(* Logix 5000 project; controller STAT 1756-L72 rev 20.12; software revision 20.04; part 13 of 34 *)
(* tags used below, declared in another part *)
   P21 : BOOL;
   P22 : BOOL;
   B14 : DINT[30];
   B16 : DINT[30];
   B17 : DINT[30];
   B3 : DINT[256];
   B9 : DINT[40];
   F8 : REAL[256];
   FL_STOP_RO : BOOL;
   I10_000_Bit00 : ALIAS FOR I10[0].0;   // Drukknop start CL7 P 19A
   I10_000_Bit01 : ALIAS FOR I10[0].1;   // Drukknop stop CL7 P 19A
   I10_000_Bit02 : ALIAS FOR I10[0].2;   // Drukknop start CL7 P 19B
   I10_000_Bit03 : ALIAS FOR I10[0].3;   // Drukknop stop CL7 P 19B
   I10_001_Bit07 : ALIAS FOR I10[1].7;   // Hand Automaat CL9
   I10_001_Bit08 : ALIAS FOR I10[1].8;   // Drukknop start P9 CL9
   I10_001_Bit09 : ALIAS FOR I10[1].9;   // Drukknop stop P7 CL9
   I10_001_Bit10 : ALIAS FOR I10[1].10;   // Drukknop start P8 CL9
   I10_001_Bit11 : ALIAS FOR I10[1].11;   // Drukknop stop P8 CL9
   I10_001_Bit12 : ALIAS FOR I10[1].12;   // Drukknop start P9 CL9
   I10_001_Bit13 : ALIAS FOR I10[1].13;   // Drukknop stop P9 CL9
   I19_000_Bit00 : ALIAS FOR I19[0].0;   // VANNE ALIBERT OUVERTE
   I19_000_Bit01 : ALIAS FOR I19[0].1;   // VANNE ALIBERT FERMEE
   I1_005_Bit15 : ALIAS FOR I1[5].15;
   I1_016_Bit06 : ALIAS FOR I1[16].6;   // CL2 start res.
   I2_000_Bit04 : ALIAS FOR I2[0].4;   // Deelnoodstop cl6 eurowater
   I2_000_Bit06 : ALIAS FOR I2[0].6;   // Deelnoodstop cl7 IBT B
   I3_000_Bit09 : ALIAS FOR I3[0].9;   // Motor pro 1 voedingpomp osmose 1 in driehoek
   I3_000_Bit10 : ALIAS FOR I3[0].10;   // Motor pro 1 voedingpomp osmose 1 in ster
   I3_000_Bit13 : ALIAS FOR I3[0].13;   // Motor pro 2 voedingpomp osmose 2 in driehoek
   I3_000_Bit14 : ALIAS FOR I3[0].14;   // Motor pro 2 voedingpomp osmose 2 in ster
   I3_001_Bit01 : ALIAS FOR I3[1].1;   // Motor p21 kuip az in driehoek
   I3_001_Bit02 : ALIAS FOR I3[1].2;   // Motor p21 kuip az in ster
   I3_001_Bit05 : ALIAS FOR I3[1].5;   // Motor p22 kuip az in driehoek
   I3_001_Bit06 : ALIAS FOR I3[1].6;   // Motor p22 kuip az in ster
   I3_001_Bit09 : ALIAS FOR I3[1].9;   // Motor voedingspomp osmose 3 in drie
   I3_001_Bit10 : ALIAS FOR I3[1].10;   // Motor voed osmose 3 ster
   I6_000_Bit10 : ALIAS FOR I6[0].10;   // pressostaat osmose1
   I6_000_Bit11 : ALIAS FOR I6[0].11;   // pressostaat osmose2
   I6_000_Bit12 : ALIAS FOR I6[0].12;   // pressostaat osmose3
   I7_000_Bit08 : ALIAS FOR I7[0].8;   // midden alarm ketel tampon
   I7_000_Bit09 : ALIAS FOR I7[0].9;   // laag alarm ketel tampon
   I8_000_Bit00 : ALIAS FOR I8[0].0;   // niveau kuip az hoog alarm
   I8_000_Bit01 : ALIAS FOR I8[0].1;   // niveau kuip az midden
   I8_000_Bit02 : ALIAS FOR I8[0].2;   // niveau kuip az laag niv
   I8_000_Bit04 : ALIAS FOR I8[0].4;   // niveau kuip 20m hoog alarm
   I8_000_Bit05 : ALIAS FOR I8[0].5;   // niveau midden kuip 20m
   I8_000_Bit06 : ALIAS FOR I8[0].6;   // niveau kuip 20m laag niv
   I8_000_Bit08 : ALIAS FOR I8[0].8;   // laag niveau kuip 1 voorb. polyelectrolute
   I8_000_Bit11 : ALIAS FOR I8[0].11;   // hoog niveau kuip 2 voorb. polyelectrolute
   I8_001_Bit09 : ALIAS FOR I8[1].9;   // Schakelaar hand autom cl6
   I8_001_Bit10 : ALIAS FOR I8[1].10;   // drukknop start cl6 pro1
   I8_001_Bit11 : ALIAS FOR I8[1].11;   // drukknop stop cl6 pro1
   I8_001_Bit12 : ALIAS FOR I8[1].12;   // drukknop start cl6 pro2
   I8_001_Bit13 : ALIAS FOR I8[1].13;   // drukknop stop cl6 pro2
   I8_001_Bit14 : ALIAS FOR I8[1].14;   // drukknop start cl6 p21
   I8_001_Bit15 : ALIAS FOR I8[1].15;   // drukknop stop cl6 p21
   I9_000_Bit00 : ALIAS FOR I9[0].0;   // Drukknop start CL6 P22
   I9_000_Bit01 : ALIAS FOR I9[0].1;   // Drukknop stop CL6 P22
   I9_000_Bit02 : ALIAS FOR I9[0].2;   // Drukknop start CL6 PRO3
   I9_000_Bit03 : ALIAS FOR I9[0].3;   // Drukknop stop CL6 PRO3
   I9_000_Bit04 : ALIAS FOR I9[0].4;   // Drukknop start CL6 P21
   I9_000_Bit05 : ALIAS FOR I9[0].5;   // Drukknop stop CL6 P21
   I9_000_Bit09 : ALIAS FOR I9[0].9;   // Hand_Auto CL7
   I9_001_Bit06 : ALIAS FOR I9[1].6;   // Drukknop start CL7 AG1
   I9_001_Bit07 : ALIAS FOR I9[1].7;   // Drukknop stop CL7 AG1
   I9_001_Bit08 : ALIAS FOR I9[1].8;   // Drukknop start CL7 AG2
   I9_001_Bit09 : ALIAS FOR I9[1].9;   // Drukknop stop CL7 AG2
   I9_001_Bit10 : ALIAS FOR I9[1].10;   // Drukknop start CL7 AG3
   I9_001_Bit11 : ALIAS FOR I9[1].11;   // Drukknop stop CL7 AG3
   N11 : DINT[150];
   N12 : DINT[230];
   N13 : DINT[230];
   O12_000_Bit03 : ALIAS FOR O12[0].3;   // motor ag1 mixer krimp neutralisatie AG1_MIXER_KRIMP
   O12_000_Bit08 : ALIAS FOR O12[0].8;   // pomp ag2 mixer vat 1 AG2_MIXER_VAT1
   O12_000_Bit09 : ALIAS FOR O12[0].9;   // pomp ag3 mixer vat 2 AG3_MIXER_VAT2
   O12_000_Bit12 : ALIAS FOR O12[0].12;   // Motor P19a zuiveringspomp controleweger P19_ZUIVERP
   O12_000_Bit13 : ALIAS FOR O12[0].13;   // Motor P20 zuiveringspomp controleweger P20_ZUIVERP
   O12_001_Bit03 : ALIAS FOR O12[1].3;   // Motor P7 voedingspomp omgekeerde osmose 1 P7_OSMOSE_1
   O12_001_Bit04 : ALIAS FOR O12[1].4;   // Motor P8 voedingspomp omgekeerde osmose 2 P8_OSMOSE_2
   O12_001_Bit05 : ALIAS FOR O12[1].5;   // Motor P9 voedingspomp omgekeerde osmose 3 P9_OSMOSE_3
   O15_001_Bit07 : ALIAS FOR O15[1].7;   // EV3 EV3
   O16_000_Bit00 : ALIAS FOR O16[0].0;   // COMMANDE VANNE ALIBERT
   O18_001_Bit00 : ALIAS FOR O18[1].0;   // pompe 1 puisard ligne 4
   O18_001_Bit01 : ALIAS FOR O18[1].1;   // pompe 2 puisard ligne 4
   O18_001_Bit06 : ALIAS FOR O18[1].6;
   O18_001_Bit07 : ALIAS FOR O18[1].7;   // pomp pompen uit kelder p23
   O18_001_Bit08 : ALIAS FOR O18[1].8;   // pomp pompen uit kelder p24
   P23 : BOOL;
   P24 : BOOL;
   T27 : TIMER[100];
   T4 : TIMER[200];
(* ibt, continued *)

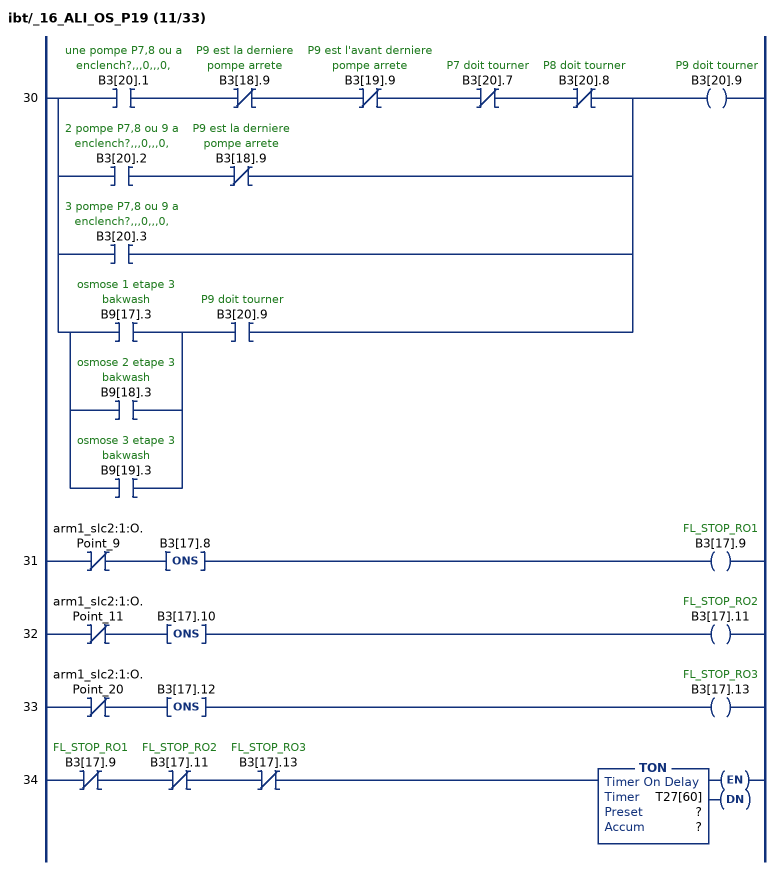
   [picture p202: ibt/_16_ALI_OS_P19 rungs 30-34]
   30: [XIC(B3[20].1) XIO(B3[18].9) XIO(B3[19].9) XIO(B3[20].7) XIO(B3[20].8) ,[XIC(B3[20].2) XIO(B3[18].9) ,XIC(B3[20].3) ] ,[XIC(B9[17].3) ,XIC(B9[18].3) ,XIC(B9[19].3) ] XIC(B3[20].9) ]OTE(B3[20].9);
   31: XIO(arm1_slc2:1:O.Point_9)ONS(B3[17].8)OTE(B3[17].9);
   32: XIO(arm1_slc2:1:O.Point_11)ONS(B3[17].10)OTE(B3[17].11);
   33: XIO(arm1_slc2:1:O.Point_20)ONS(B3[17].12)OTE(B3[17].13);
   34: XIO(B3[17].9)XIO(B3[17].11)XIO(B3[17].13)TON(T27[60],?,?);
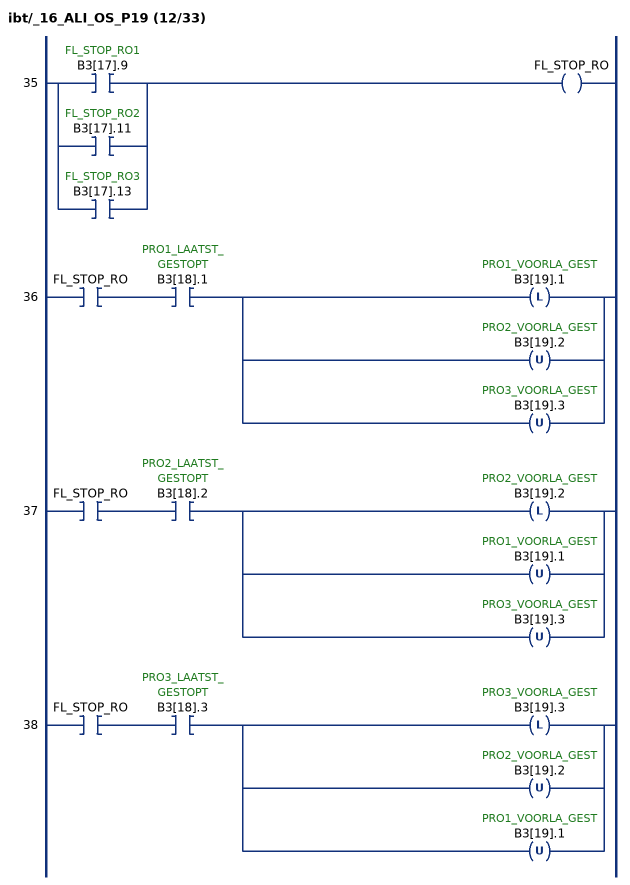
   35: [XIC(B3[17].9) ,[XIC(B3[17].11) ,XIC(B3[17].13) ] ]OTE(FL_STOP_RO);
   36: XIC(FL_STOP_RO)XIC(B3[18].1)[OTL(B3[19].1) ,[OTU(B3[19].2) ,OTU(B3[19].3) ] ];
   37: XIC(FL_STOP_RO)XIC(B3[18].2)[OTL(B3[19].2) ,[OTU(B3[19].1) ,OTU(B3[19].3) ] ];
   38: XIC(FL_STOP_RO)XIC(B3[18].3)[OTL(B3[19].3) ,[OTU(B3[19].2) ,OTU(B3[19].1) ] ];
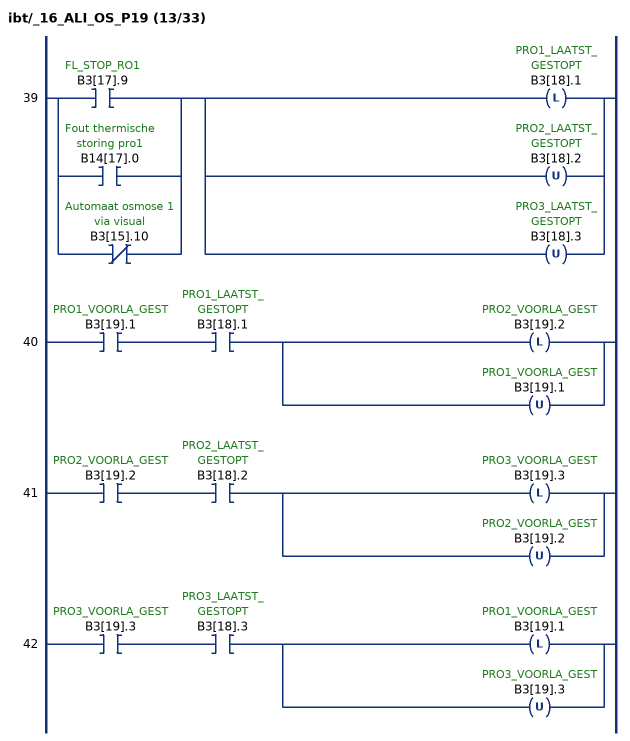
   39: [XIC(B3[17].9) ,[XIC(B14[17].0) ,XIO(B3[15].10) ] ][OTL(B3[18].1) ,[OTU(B3[18].2) ,OTU(B3[18].3) ] ];
   40: XIC(B3[19].1)XIC(B3[18].1)[OTL(B3[19].2) ,OTU(B3[19].1) ];
   41: XIC(B3[19].2)XIC(B3[18].2)[OTL(B3[19].3) ,OTU(B3[19].2) ];
   42: XIC(B3[19].3)XIC(B3[18].3)[OTL(B3[19].1) ,OTU(B3[19].3) ];
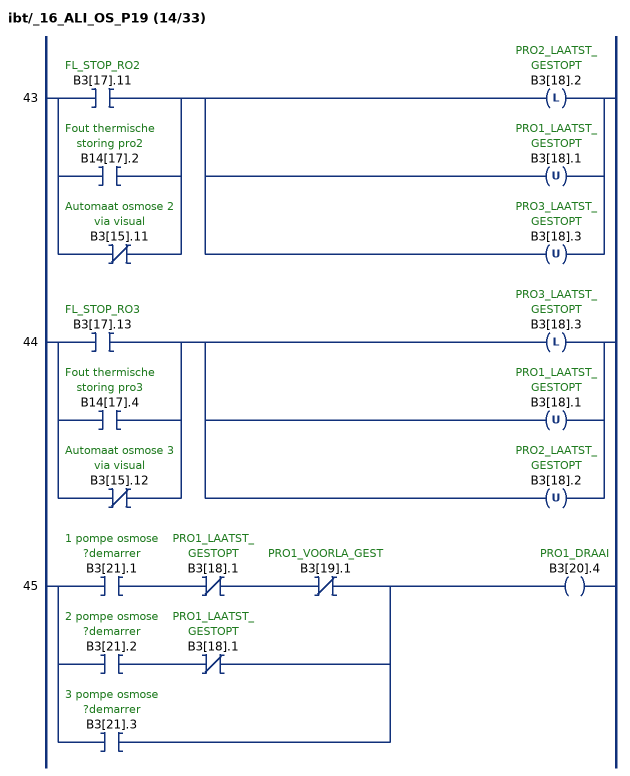
   43: [XIC(B3[17].11) ,[XIC(B14[17].2) ,XIO(B3[15].11) ] ][OTL(B3[18].2) ,[OTU(B3[18].1) ,OTU(B3[18].3) ] ];
   44: [XIC(B3[17].13) ,[XIC(B14[17].4) ,XIO(B3[15].12) ] ][OTL(B3[18].3) ,[OTU(B3[18].1) ,OTU(B3[18].2) ] ];
   45: [XIC(B3[21].1) XIO(B3[18].1) XIO(B3[19].1) ,[XIC(B3[21].2) XIO(B3[18].1) ,XIC(B3[21].3) ] ]OTE(B3[20].4);
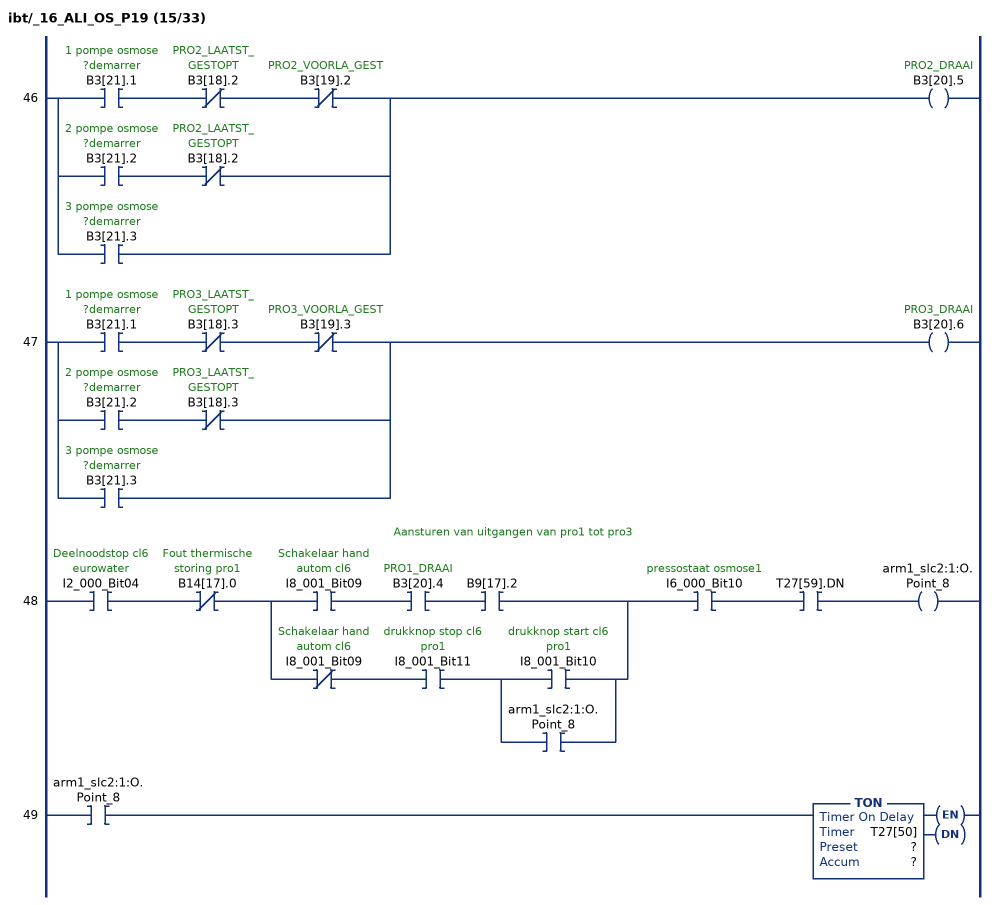
   46: [XIC(B3[21].1) XIO(B3[18].2) XIO(B3[19].2) ,[XIC(B3[21].2) XIO(B3[18].2) ,XIC(B3[21].3) ] ]OTE(B3[20].5);
   47: [XIC(B3[21].1) XIO(B3[18].3) XIO(B3[19].3) ,[XIC(B3[21].2) XIO(B3[18].3) ,XIC(B3[21].3) ] ]OTE(B3[20].6);
   // Aansturen van uitgangen van pro1 tot pro3
   48: XIC(I2_000_Bit04)XIO(B14[17].0)[XIC(I8_001_Bit09) XIC(B3[20].4) XIC(B9[17].2) ,XIO(I8_001_Bit09) XIC(I8_001_Bit11) [XIC(I8_001_Bit10) ,XIC(arm1_slc2:1:O.Point_8) ] ]XIC(I6_000_Bit10)XIC(T27[59].DN)OTE(arm1_slc2:1:O.Point_8);
   49: XIC(arm1_slc2:1:O.Point_8)TON(T27[50],?,?);
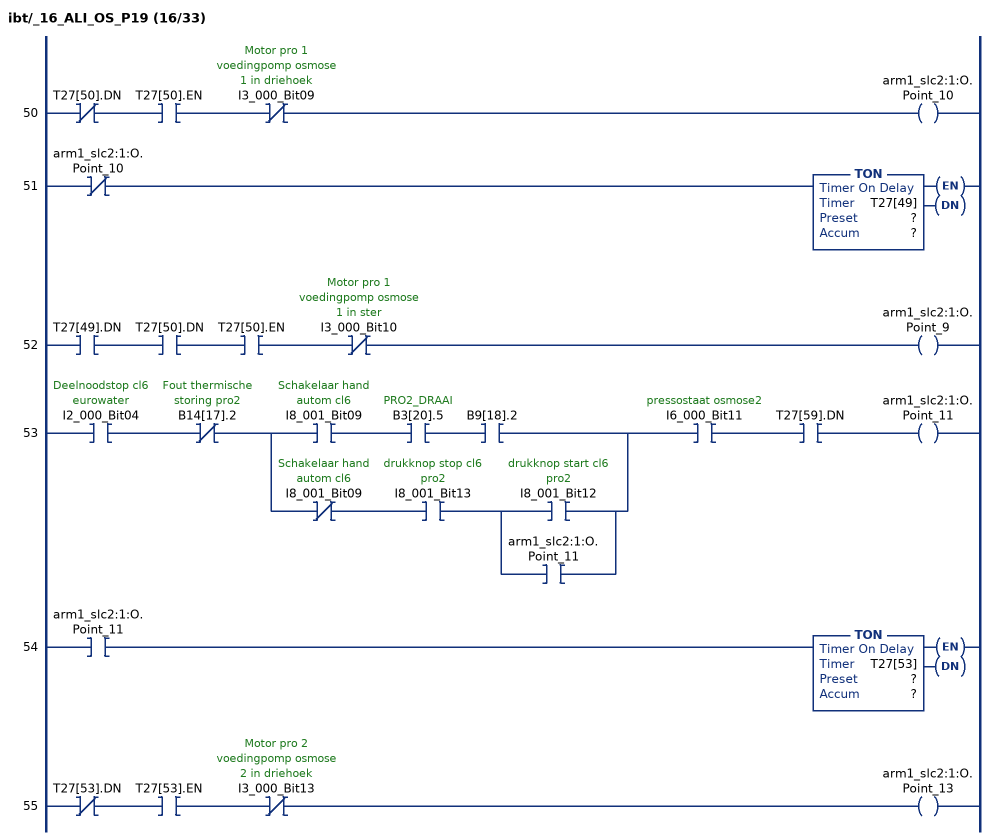
   50: XIO(T27[50].DN)XIC(T27[50].EN)XIO(I3_000_Bit09)OTE(arm1_slc2:1:O.Point_10);
   51: XIO(arm1_slc2:1:O.Point_10)TON(T27[49],?,?);
   52: XIC(T27[49].DN)XIC(T27[50].DN)XIC(T27[50].EN)XIO(I3_000_Bit10)OTE(arm1_slc2:1:O.Point_9);
   53: XIC(I2_000_Bit04)XIO(B14[17].2)[XIC(I8_001_Bit09) XIC(B3[20].5) XIC(B9[18].2) ,XIO(I8_001_Bit09) XIC(I8_001_Bit13) [XIC(I8_001_Bit12) ,XIC(arm1_slc2:1:O.Point_11) ] ]XIC(I6_000_Bit11)XIC(T27[59].DN)OTE(arm1_slc2:1:O.Point_11);
   54: XIC(arm1_slc2:1:O.Point_11)TON(T27[53],?,?);
   55: XIO(T27[53].DN)XIC(T27[53].EN)XIO(I3_000_Bit13)OTE(arm1_slc2:1:O.Point_13);
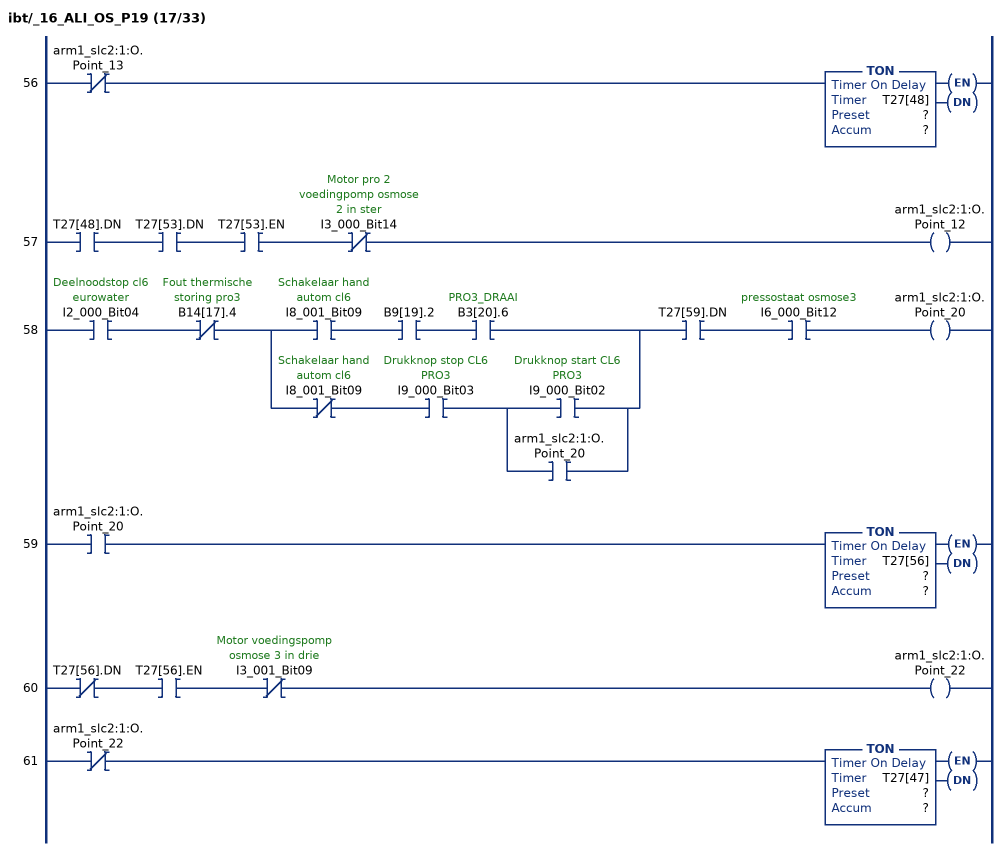
   56: XIO(arm1_slc2:1:O.Point_13)TON(T27[48],?,?);
   57: XIC(T27[48].DN)XIC(T27[53].DN)XIC(T27[53].EN)XIO(I3_000_Bit14)OTE(arm1_slc2:1:O.Point_12);
   58: XIC(I2_000_Bit04)XIO(B14[17].4)[XIC(I8_001_Bit09) XIC(B9[19].2) XIC(B3[20].6) ,XIO(I8_001_Bit09) XIC(I9_000_Bit03) [XIC(I9_000_Bit02) ,XIC(arm1_slc2:1:O.Point_20) ] ]XIC(T27[59].DN)XIC(I6_000_Bit12)OTE(arm1_slc2:1:O.Point_20);
   59: XIC(arm1_slc2:1:O.Point_20)TON(T27[56],?,?);
   60: XIO(T27[56].DN)XIC(T27[56].EN)XIO(I3_001_Bit09)OTE(arm1_slc2:1:O.Point_22);
   61: XIO(arm1_slc2:1:O.Point_22)TON(T27[47],?,?);
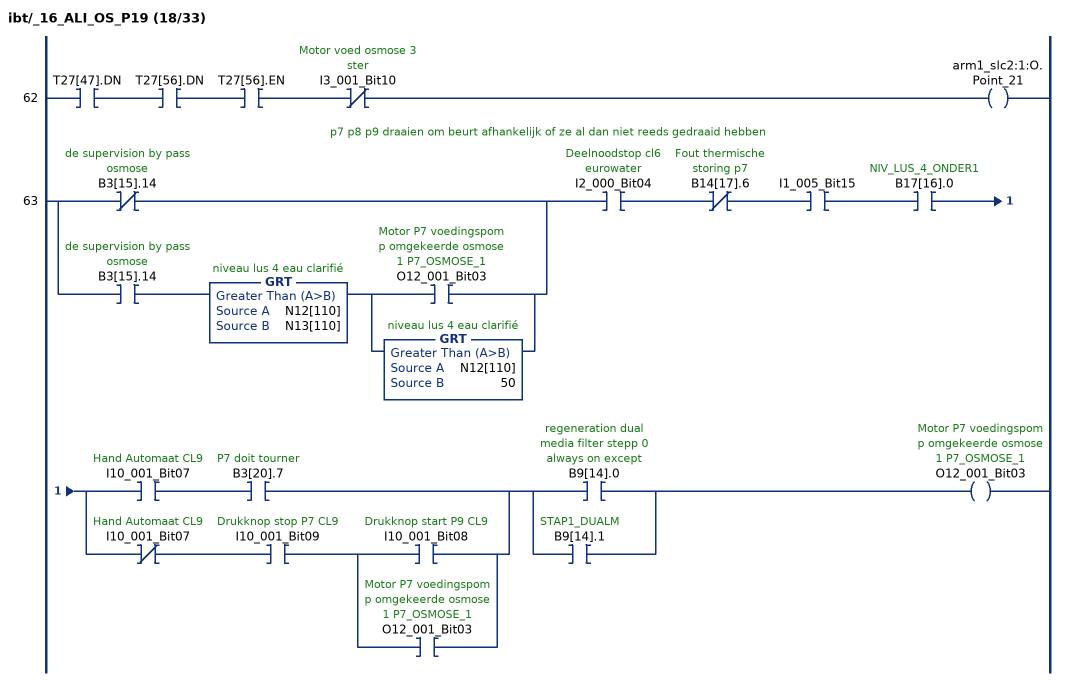
   62: XIC(T27[47].DN)XIC(T27[56].DN)XIC(T27[56].EN)XIO(I3_001_Bit10)OTE(arm1_slc2:1:O.Point_21);
   // p7 p8 p9 draaien om beurt afhankelijk of ze al dan niet reeds gedraaid hebben
   63: [XIO(B3[15].14) ,XIC(B3[15].14) GRT(N12[110],N13[110]) [XIC(O12_001_Bit03) ,GRT(N12[110],50) ] ]XIC(I2_000_Bit04)XIO(B14[17].6)XIC(I1_005_Bit15)XIC(B17[16].0)[XIC(I10_001_Bit07) XIC(B3[20].7) ,XIO(I10_001_Bit07) XIC(I10_001_Bit09) [XIC(I10_001_Bit08) ,XIC(O12_001_Bit03) ] ][XIC(B9[14].0) ,XIC(B9[14].1) ]OTE(O12_001_Bit03);
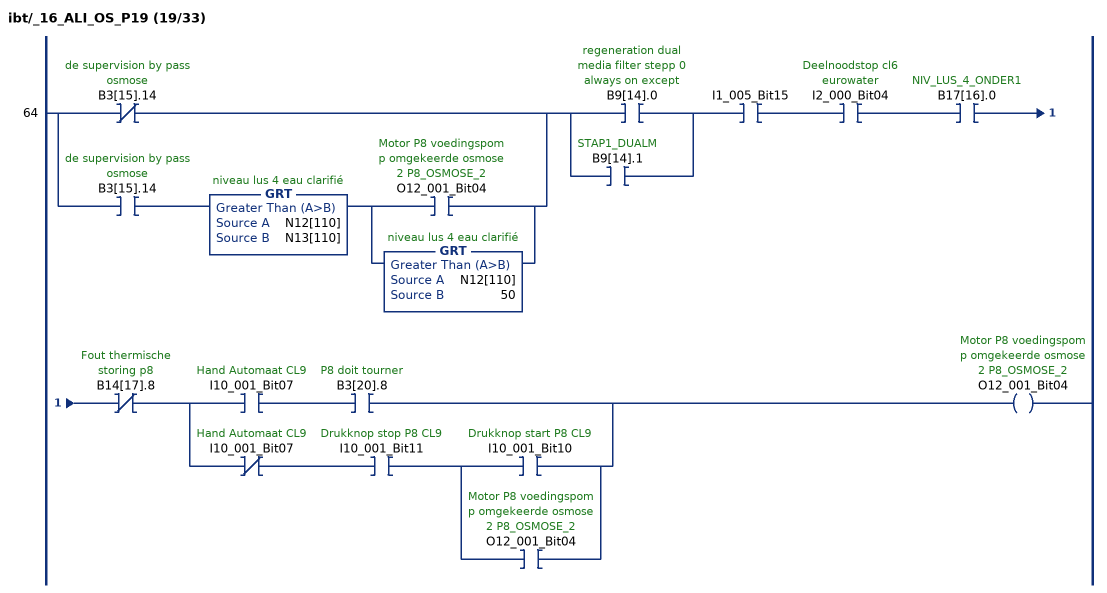
   64: [XIO(B3[15].14) ,XIC(B3[15].14) GRT(N12[110],N13[110]) [XIC(O12_001_Bit04) ,GRT(N12[110],50) ] ][XIC(B9[14].0) ,XIC(B9[14].1) ]XIC(I1_005_Bit15)XIC(I2_000_Bit04)XIC(B17[16].0)XIO(B14[17].8)[XIC(I10_001_Bit07) XIC(B3[20].8) ,XIO(I10_001_Bit07) XIC(I10_001_Bit11) [XIC(I10_001_Bit10) ,XIC(O12_001_Bit04) ] ]OTE(O12_001_Bit04);
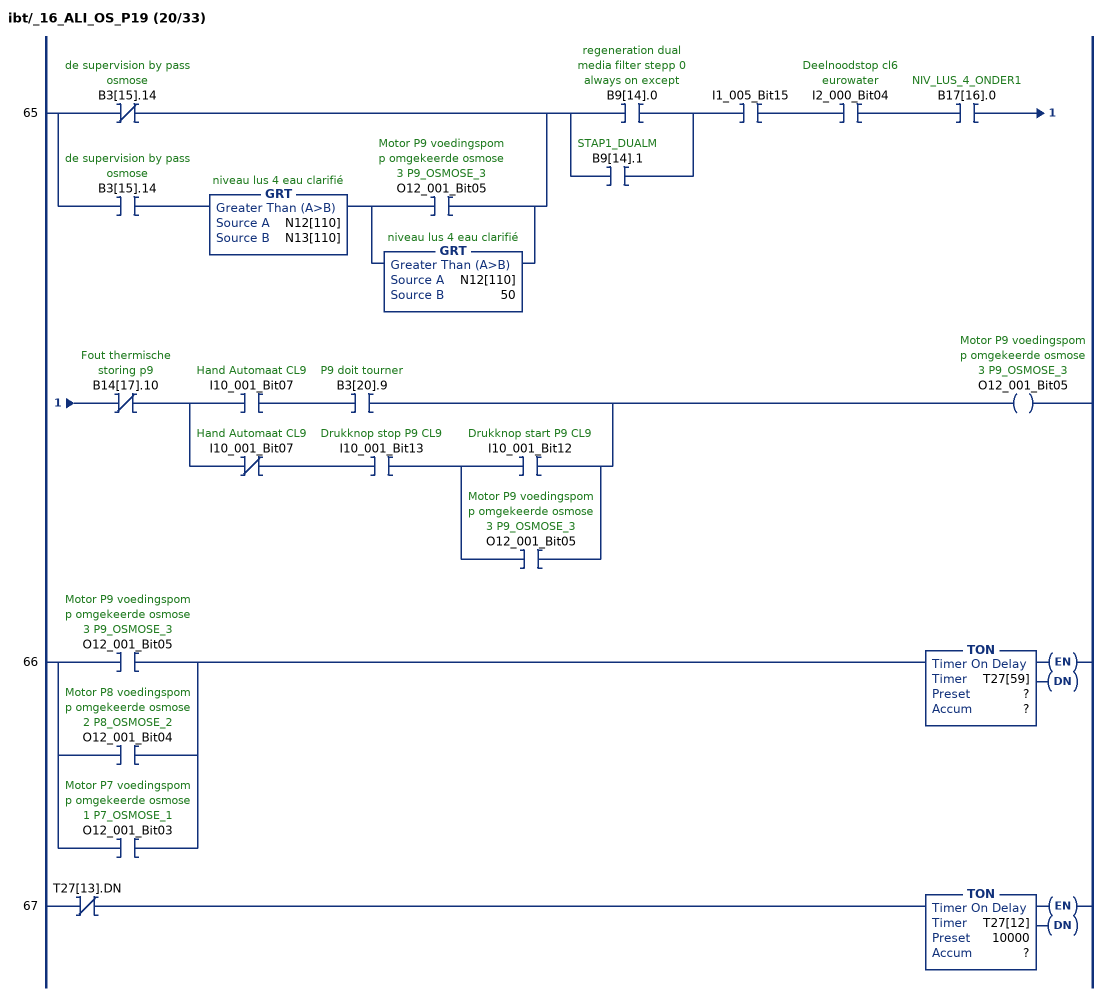
   65: [XIO(B3[15].14) ,XIC(B3[15].14) GRT(N12[110],N13[110]) [XIC(O12_001_Bit05) ,GRT(N12[110],50) ] ][XIC(B9[14].0) ,XIC(B9[14].1) ]XIC(I1_005_Bit15)XIC(I2_000_Bit04)XIC(B17[16].0)XIO(B14[17].10)[XIC(I10_001_Bit07) XIC(B3[20].9) ,XIO(I10_001_Bit07) XIC(I10_001_Bit13) [XIC(I10_001_Bit12) ,XIC(O12_001_Bit05) ] ]OTE(O12_001_Bit05);
   66: [XIC(O12_001_Bit05) ,[XIC(O12_001_Bit04) ,XIC(O12_001_Bit03) ] ]TON(T27[59],?,?);
   67: XIO(T27[13].DN)TON(T27[12],?,?);
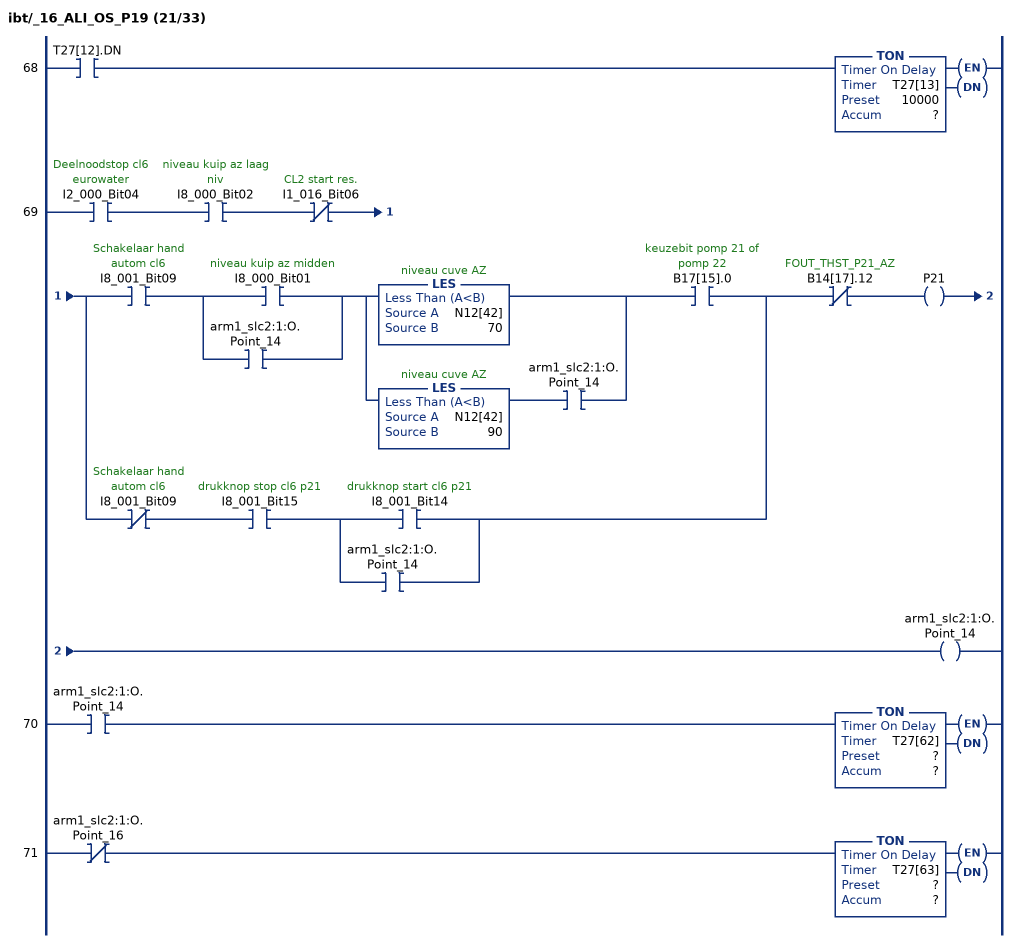
   68: XIC(T27[12].DN)TON(T27[13],?,?);
   69: XIC(I2_000_Bit04)XIC(I8_000_Bit02)XIO(I1_016_Bit06)[XIC(I8_001_Bit09) [XIC(I8_000_Bit01) ,XIC(arm1_slc2:1:O.Point_14) ] [LES(N12[42],70) ,LES(N12[42],90) XIC(arm1_slc2:1:O.Point_14) ] XIC(B17[15].0) ,XIO(I8_001_Bit09) XIC(I8_001_Bit15) [XIC(I8_001_Bit14) ,XIC(arm1_slc2:1:O.Point_14) ] ]XIO(B14[17].12)OTE(P21)OTE(arm1_slc2:1:O.Point_14);
   70: XIC(arm1_slc2:1:O.Point_14)TON(T27[62],?,?);
   71: XIO(arm1_slc2:1:O.Point_16)TON(T27[63],?,?);
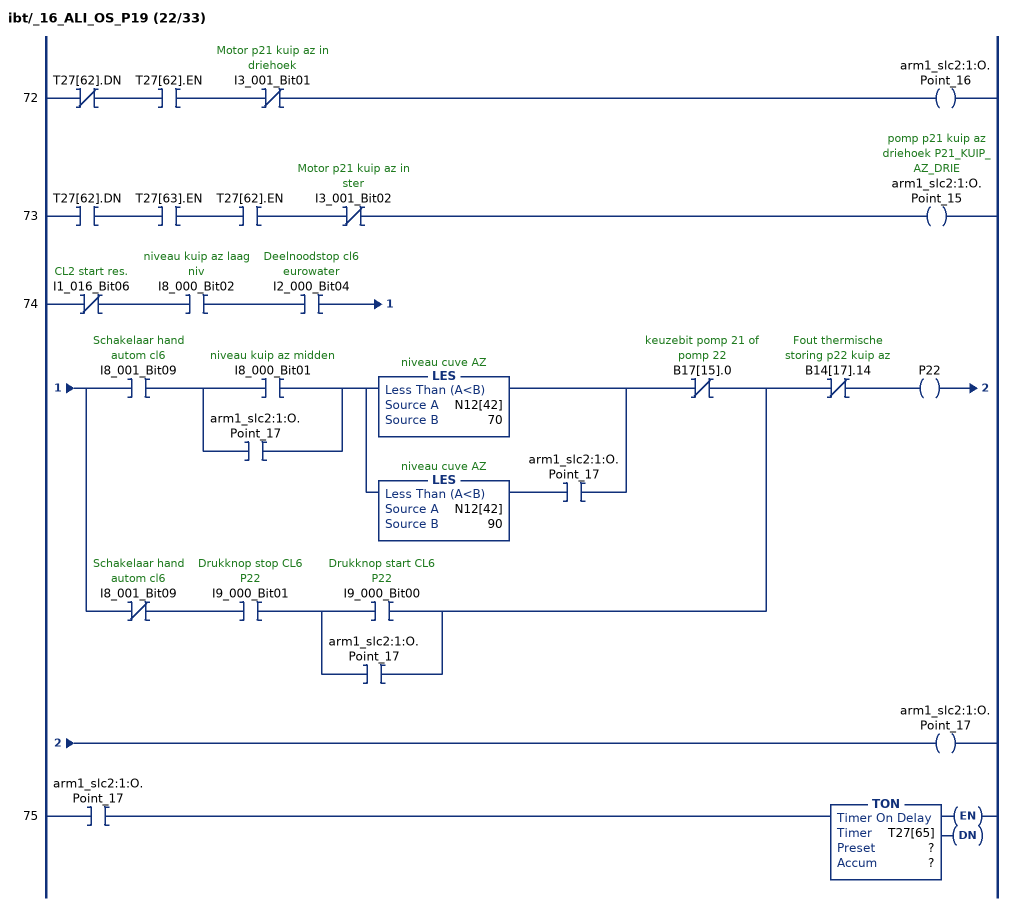
   72: XIO(T27[62].DN)XIC(T27[62].EN)XIO(I3_001_Bit01)OTE(arm1_slc2:1:O.Point_16);
   73: XIC(T27[62].DN)XIC(T27[63].EN)XIC(T27[62].EN)XIO(I3_001_Bit02)OTE(arm1_slc2:1:O.Point_15);
   74: XIO(I1_016_Bit06)XIC(I8_000_Bit02)XIC(I2_000_Bit04)[XIC(I8_001_Bit09) [XIC(I8_000_Bit01) ,XIC(arm1_slc2:1:O.Point_17) ] [LES(N12[42],70) ,LES(N12[42],90) XIC(arm1_slc2:1:O.Point_17) ] XIO(B17[15].0) ,XIO(I8_001_Bit09) XIC(I9_000_Bit01) [XIC(I9_000_Bit00) ,XIC(arm1_slc2:1:O.Point_17) ] ]XIO(B14[17].14)OTE(P22)OTE(arm1_slc2:1:O.Point_17);
   75: XIC(arm1_slc2:1:O.Point_17)TON(T27[65],?,?);
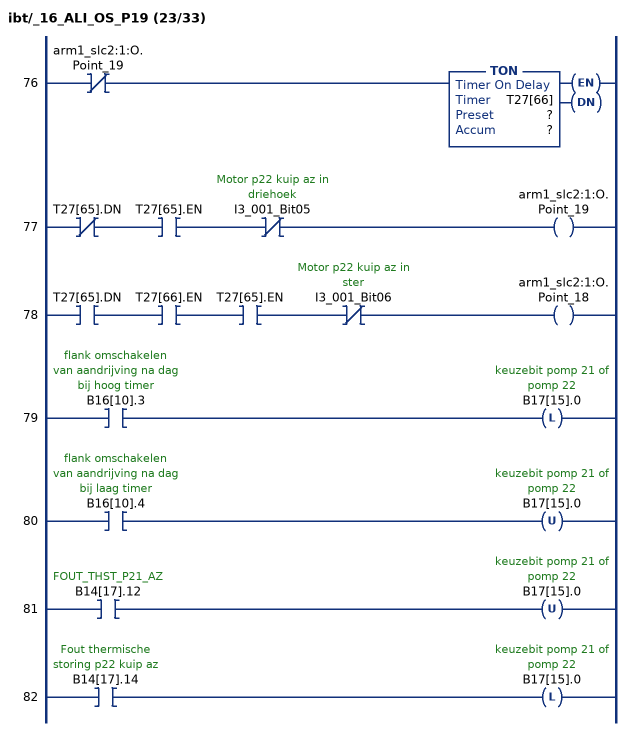
   76: XIO(arm1_slc2:1:O.Point_19)TON(T27[66],?,?);
   77: XIO(T27[65].DN)XIC(T27[65].EN)XIO(I3_001_Bit05)OTE(arm1_slc2:1:O.Point_19);
   78: XIC(T27[65].DN)XIC(T27[66].EN)XIC(T27[65].EN)XIO(I3_001_Bit06)OTE(arm1_slc2:1:O.Point_18);
   79: XIC(B16[10].3)OTL(B17[15].0);
   80: XIC(B16[10].4)OTU(B17[15].0);
   81: XIC(B14[17].12)OTU(B17[15].0);
   82: XIC(B14[17].14)OTL(B17[15].0);
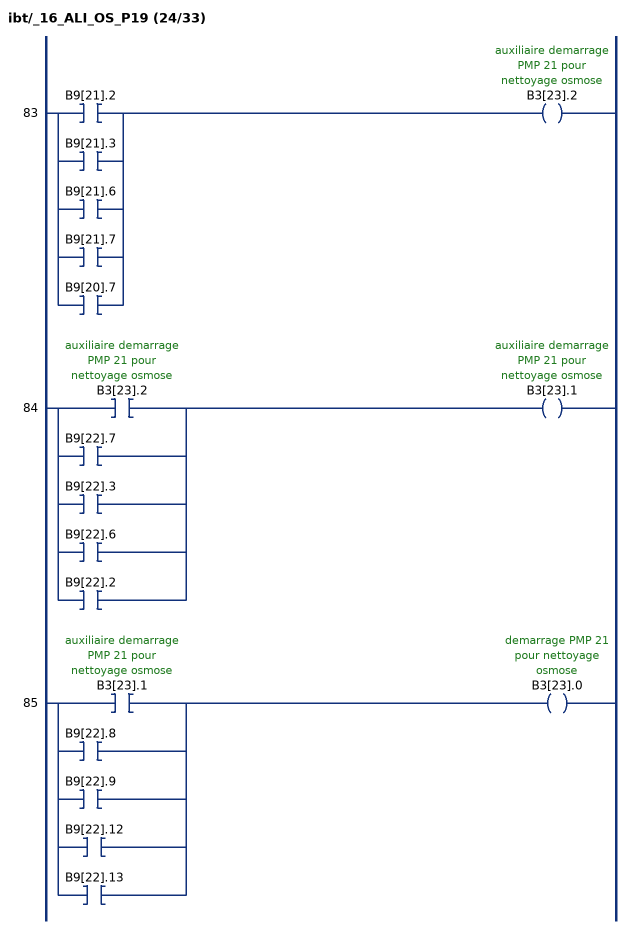
   83: [XIC(B9[21].2) ,XIC(B9[21].3) ,XIC(B9[21].6) ,XIC(B9[21].7) ,XIC(B9[20].7) ]OTE(B3[23].2);
   84: [XIC(B3[23].2) ,XIC(B9[22].7) ,XIC(B9[22].3) ,XIC(B9[22].6) ,XIC(B9[22].2) ]OTE(B3[23].1);
   85: [XIC(B3[23].1) ,XIC(B9[22].8) ,XIC(B9[22].9) ,XIC(B9[22].12) ,XIC(B9[22].13) ]OTE(B3[23].0);
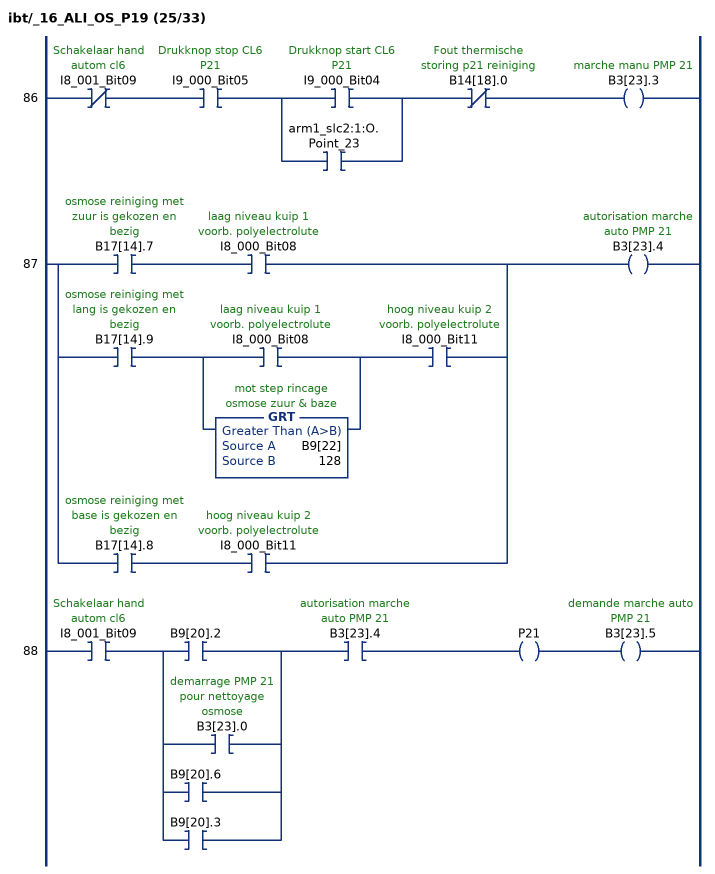
   86: XIO(I8_001_Bit09)XIC(I9_000_Bit05)[XIC(I9_000_Bit04) ,XIC(arm1_slc2:1:O.Point_23) ]XIO(B14[18].0)OTE(B3[23].3);
   87: [XIC(B17[14].7) XIC(I8_000_Bit08) ,XIC(B17[14].9) [XIC(I8_000_Bit08) ,GRT(B9[22],128) ] XIC(I8_000_Bit11) ,XIC(B17[14].8) XIC(I8_000_Bit11) ]OTE(B3[23].4);
   88: XIC(I8_001_Bit09)[XIC(B9[20].2) ,XIC(B3[23].0) ,XIC(B9[20].6) ,XIC(B9[20].3) ]XIC(B3[23].4)OTE(P21)OTE(B3[23].5);
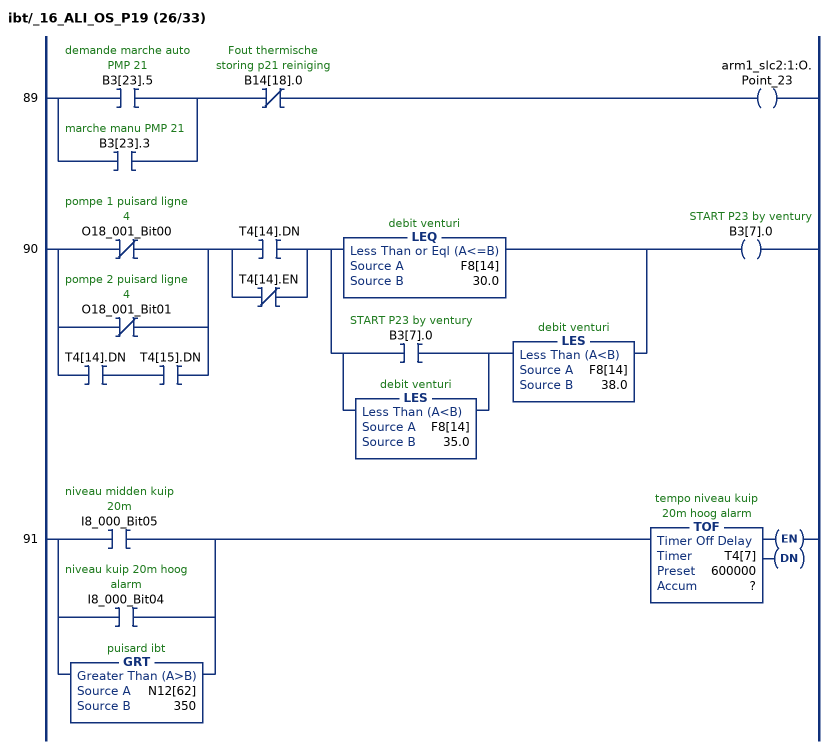
   89: [XIC(B3[23].5) ,XIC(B3[23].3) ]XIO(B14[18].0)OTE(arm1_slc2:1:O.Point_23);
   90: [XIO(O18_001_Bit00) ,XIO(O18_001_Bit01) ,XIC(T4[14].DN) XIC(T4[15].DN) ][XIC(T4[14].DN) ,XIO(T4[14].EN) ][LEQ(F8[14],30.0) ,[XIC(B3[7].0) ,LES(F8[14],35.0) ] LES(F8[14],38.0) ]OTE(B3[7].0);
   91: [XIC(I8_000_Bit05) ,XIC(I8_000_Bit04) ,GRT(N12[62],350) ]TOF(T4[7],?,?);
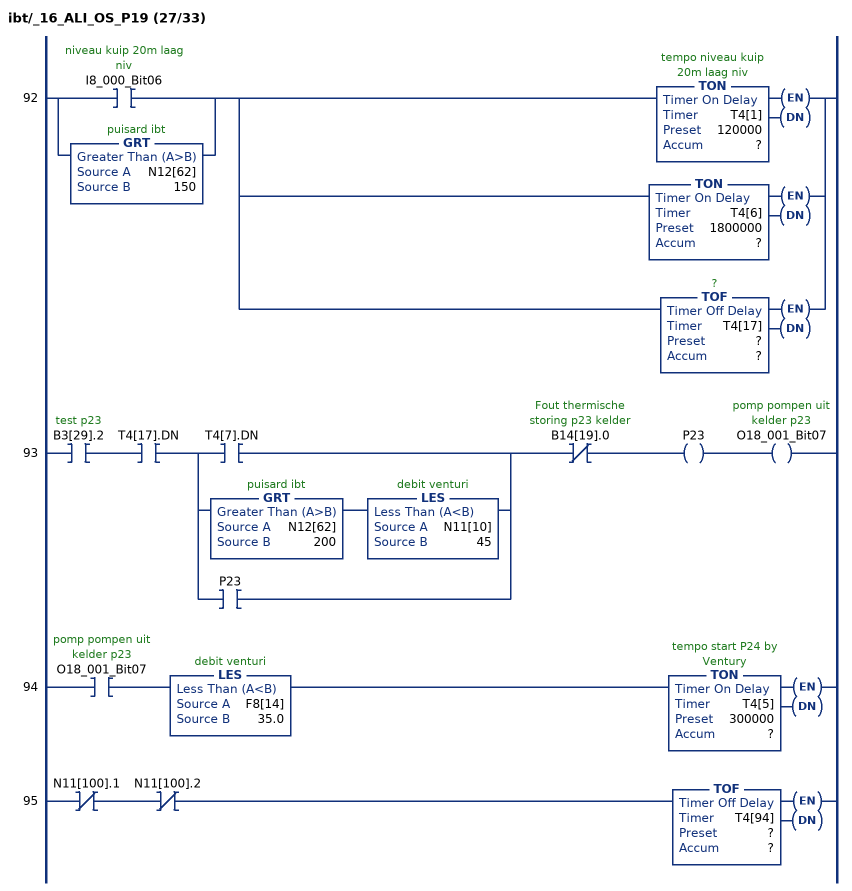
   92: [XIC(I8_000_Bit06) ,GRT(N12[62],150) ][TON(T4[1],?,?) ,TON(T4[6],?,?) ,TOF(T4[17],?,?) ];
   93: XIC(B3[29].2)XIC(T4[17].DN)[XIC(T4[7].DN) ,GRT(N12[62],200) LES(N11[10],45) ,XIC(P23) ]XIO(B14[19].0)OTE(P23)OTE(O18_001_Bit07);
   94: XIC(O18_001_Bit07)LES(F8[14],35.0)TON(T4[5],?,?);
   95: XIO(N11[100].1)XIO(N11[100].2)TOF(T4[94],?,?);
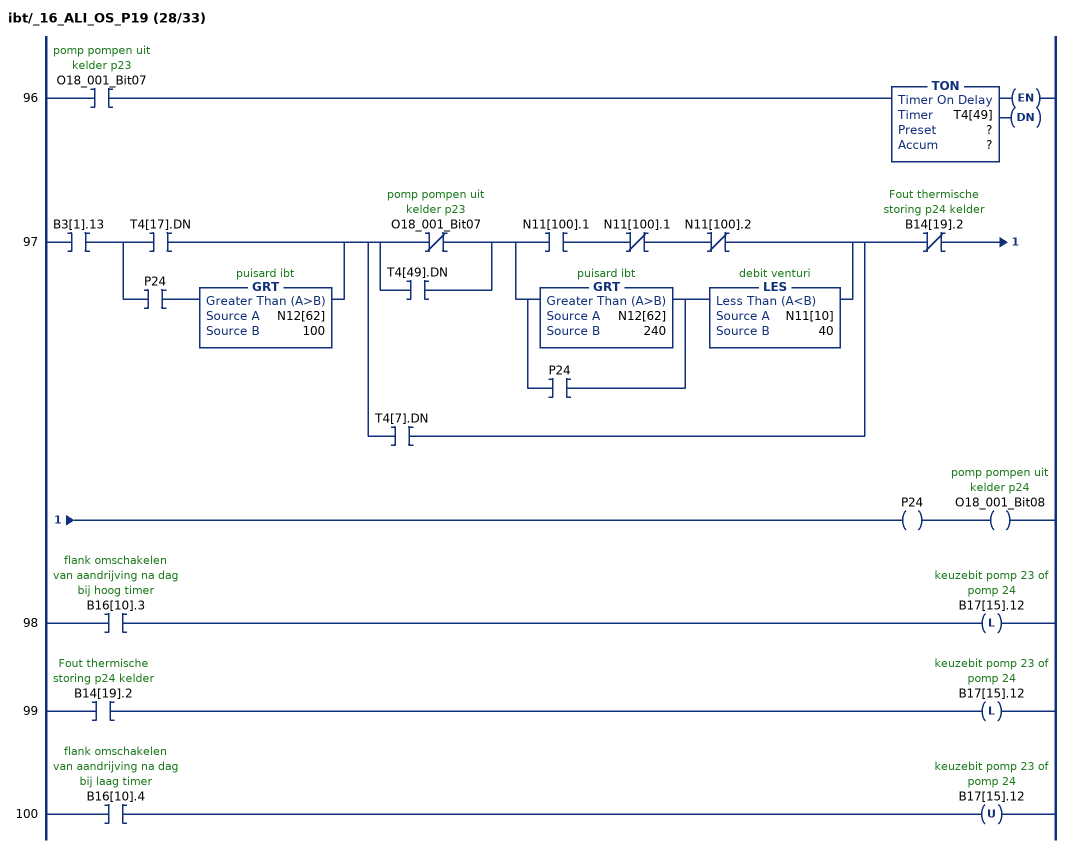
   96: XIC(O18_001_Bit07)TON(T4[49],?,?);
   97: XIC(B3[1].13)[XIC(T4[17].DN) ,XIC(P24) GRT(N12[62],100) ][[XIO(O18_001_Bit07) ,XIC(T4[49].DN) ] [XIC(N11[100].1) XIO(N11[100].1) XIO(N11[100].2) ,[GRT(N12[62],240) ,XIC(P24) ] LES(N11[10],40) ] ,XIC(T4[7].DN) ]XIO(B14[19].2)OTE(P24)OTE(O18_001_Bit08);
   98: XIC(B16[10].3)OTL(B17[15].12);
   99: XIC(B14[19].2)OTL(B17[15].12);
   100: XIC(B16[10].4)OTU(B17[15].12);
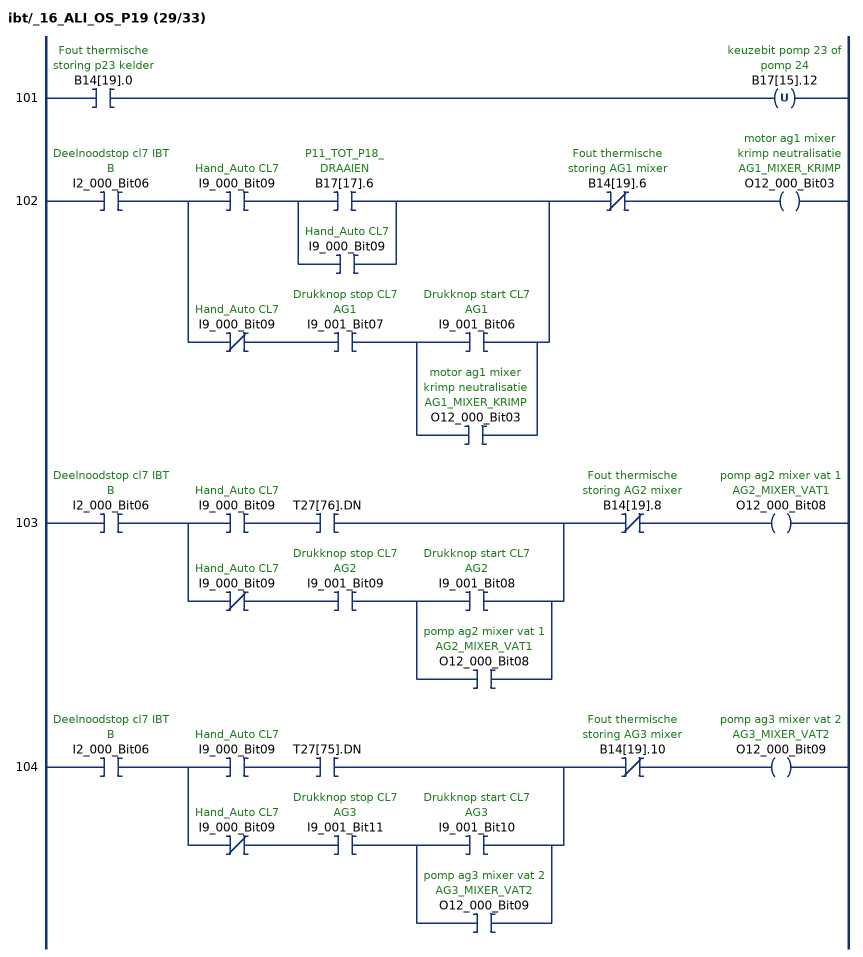
   101: XIC(B14[19].0)OTU(B17[15].12);
   102: XIC(I2_000_Bit06)[XIC(I9_000_Bit09) [XIC(B17[17].6) ,XIC(I9_000_Bit09) ] ,XIO(I9_000_Bit09) XIC(I9_001_Bit07) [XIC(I9_001_Bit06) ,XIC(O12_000_Bit03) ] ]XIO(B14[19].6)OTE(O12_000_Bit03);
   103: XIC(I2_000_Bit06)[XIC(I9_000_Bit09) XIC(T27[76].DN) ,XIO(I9_000_Bit09) XIC(I9_001_Bit09) [XIC(I9_001_Bit08) ,XIC(O12_000_Bit08) ] ]XIO(B14[19].8)OTE(O12_000_Bit08);
   104: XIC(I2_000_Bit06)[XIC(I9_000_Bit09) XIC(T27[75].DN) ,XIO(I9_000_Bit09) XIC(I9_001_Bit11) [XIC(I9_001_Bit10) ,XIC(O12_000_Bit09) ] ]XIO(B14[19].10)OTE(O12_000_Bit09);
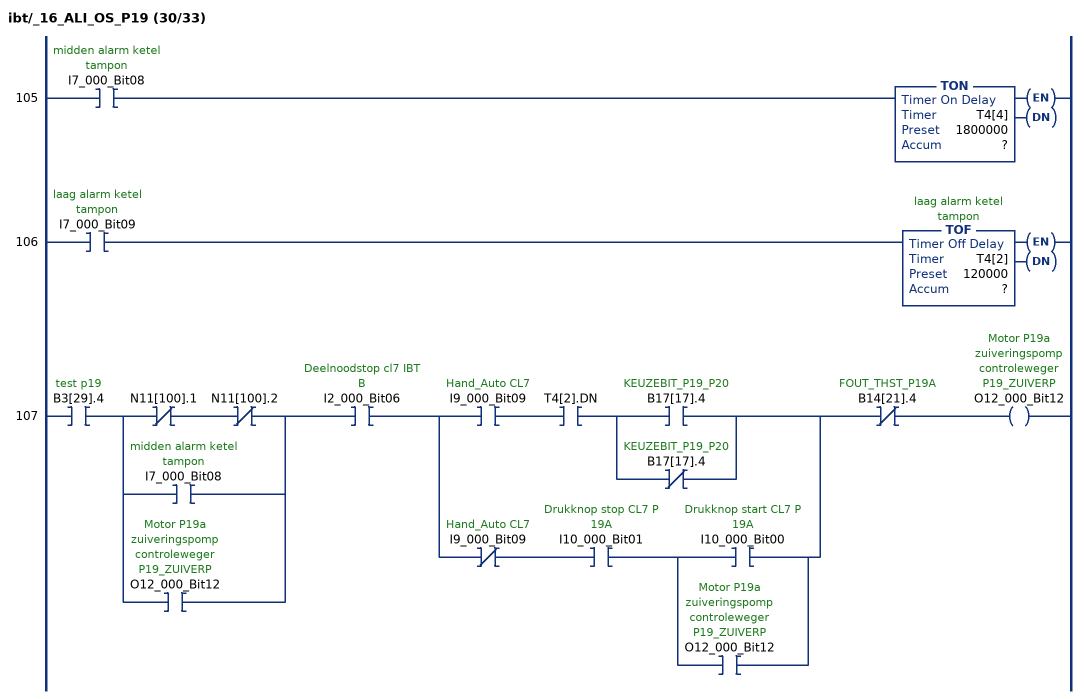
   105: XIC(I7_000_Bit08)TON(T4[4],?,?);
   106: XIC(I7_000_Bit09)TOF(T4[2],?,?);
   107: XIC(B3[29].4)[XIO(N11[100].1) XIO(N11[100].2) ,XIC(I7_000_Bit08) ,XIC(O12_000_Bit12) ]XIC(I2_000_Bit06)[XIC(I9_000_Bit09) XIC(T4[2].DN) [XIC(B17[17].4) ,XIO(B17[17].4) ] ,XIO(I9_000_Bit09) XIC(I10_000_Bit01) [XIC(I10_000_Bit00) ,XIC(O12_000_Bit12) ] ]XIO(B14[21].4)OTE(O12_000_Bit12);
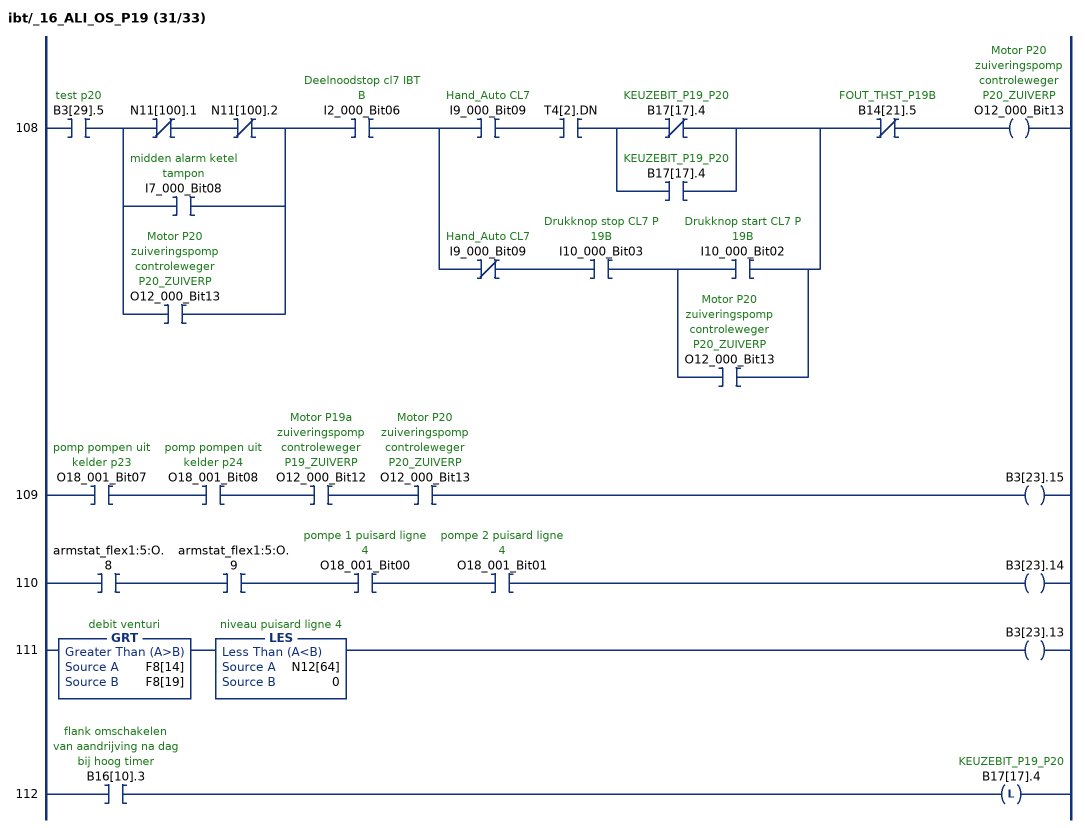
   108: XIC(B3[29].5)[XIO(N11[100].1) XIO(N11[100].2) ,XIC(I7_000_Bit08) ,XIC(O12_000_Bit13) ]XIC(I2_000_Bit06)[XIC(I9_000_Bit09) XIC(T4[2].DN) [XIO(B17[17].4) ,XIC(B17[17].4) ] ,XIO(I9_000_Bit09) XIC(I10_000_Bit03) [XIC(I10_000_Bit02) ,XIC(O12_000_Bit13) ] ]XIO(B14[21].5)OTE(O12_000_Bit13);
   109: XIC(O18_001_Bit07)XIC(O18_001_Bit08)XIC(O12_000_Bit12)XIC(O12_000_Bit13)OTE(B3[23].15);
   110: XIC(armstat_flex1:5:O.8)XIC(armstat_flex1:5:O.9)XIC(O18_001_Bit00)XIC(O18_001_Bit01)OTE(B3[23].14);
   111: GRT(F8[14],F8[19])LES(N12[64],0)OTE(B3[23].13);
   112: XIC(B16[10].3)OTL(B17[17].4);
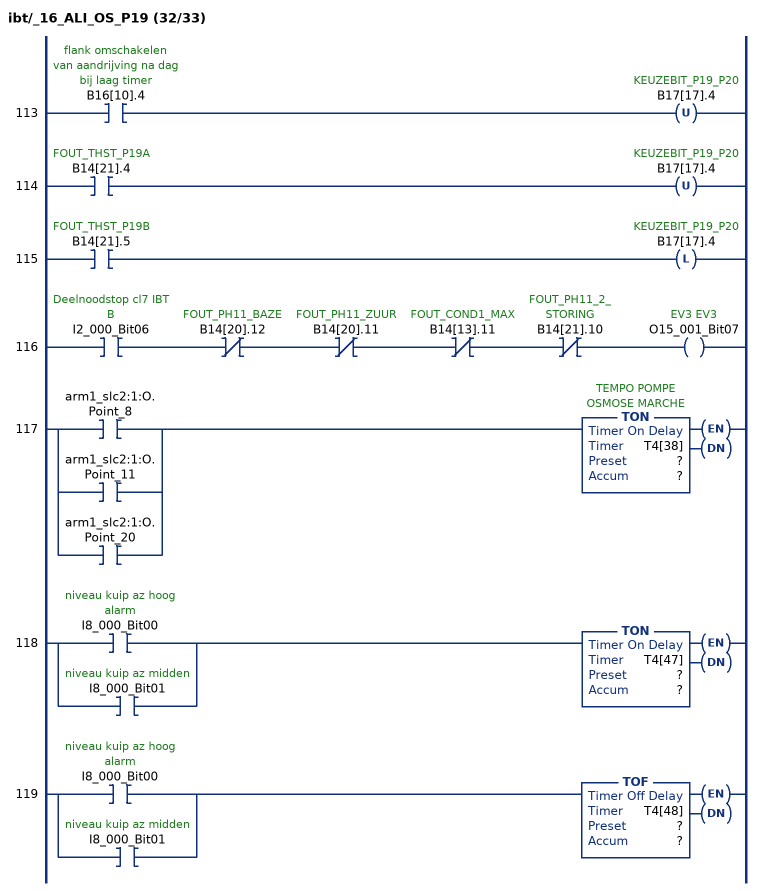
   113: XIC(B16[10].4)OTU(B17[17].4);
   114: XIC(B14[21].4)OTU(B17[17].4);
   115: XIC(B14[21].5)OTL(B17[17].4);
   116: XIC(I2_000_Bit06)XIO(B14[20].12)XIO(B14[20].11)XIO(B14[13].11)XIO(B14[21].10)OTE(O15_001_Bit07);
   117: [XIC(arm1_slc2:1:O.Point_8) ,XIC(arm1_slc2:1:O.Point_11) ,XIC(arm1_slc2:1:O.Point_20) ]TON(T4[38],?,?);
   118: [XIC(I8_000_Bit00) ,XIC(I8_000_Bit01) ]TON(T4[47],?,?);
   119: [XIC(I8_000_Bit00) ,XIC(I8_000_Bit01) ]TOF(T4[48],?,?);
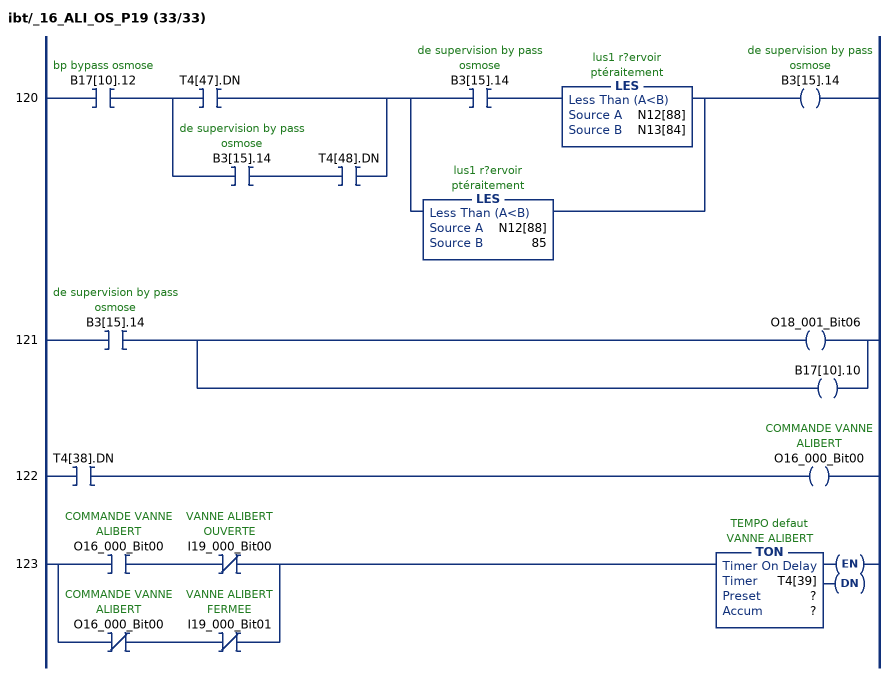
   120: XIC(B17[10].12)[XIC(T4[47].DN) ,XIC(B3[15].14) XIC(T4[48].DN) ][XIC(B3[15].14) LES(N12[88],N13[84]) ,LES(N12[88],85) ]OTE(B3[15].14);
   121: XIC(B3[15].14)[OTE(O18_001_Bit06) ,OTE(B17[10].10) ];
   122: XIC(T4[38].DN)OTE(O16_000_Bit00);
   123: [XIC(O16_000_Bit00) XIO(I19_000_Bit00) ,XIO(O16_000_Bit00) XIO(I19_000_Bit01) ]TON(T4[39],?,?);
END_ROUTINE
